ADAPTER eGenAdapter (* Adapter Interface *)
  (* Standard: 61499-1 *)
  (* Version 1.0, 2025-05-05, Maximilian Scharf *)
  SERVICE PLUG/SOCKET
    SEQUENCE request_confirm
      SOCKET.REQ(REQD) -> PLUG.REQ(REQD);
      PLUG.CNF(CNFD) -> SOCKET.CNF(CNFD);
    END_SEQUENCE
    SEQUENCE indication_response
      PLUG.IND(INDD) -> SOCKET.IND(INDD);
      SOCKET.RSP(RSPD) -> PLUG.RSP(RSPD);
    END_SEQUENCE
  END_SERVICE
END_ADAPTER
